// Mitsubishi GX Works2 project: FLASH_EX   PLC: Q03UDV

PROGRAM MAIN
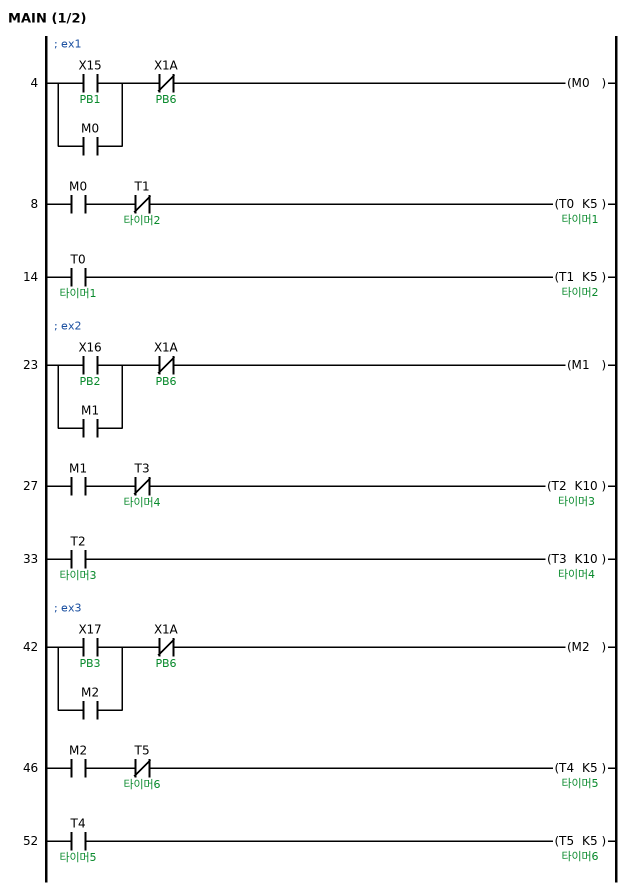
; ex1
4     LD      X15  ; PB1
      OR      M0
      ANI     X1A  ; PB6
      OUT     M0
8     LD      M0
      ANI     T1  ; 타이머2
      OUT     T0 K5  ; 타이머1
14    LD      T0  ; 타이머1
      OUT     T1 K5  ; 타이머2
; ex2
23    LD      X16  ; PB2
      OR      M1
      ANI     X1A  ; PB6
      OUT     M1
27    LD      M1
      ANI     T3  ; 타이머4
      OUT     T2 K10  ; 타이머3
33    LD      T2  ; 타이머3
      OUT     T3 K10  ; 타이머4
; ex3
42    LD      X17  ; PB3
      OR      M2
      ANI     X1A  ; PB6
      OUT     M2
46    LD      M2
      ANI     T5  ; 타이머6
      OUT     T4 K5  ; 타이머5
52    LD      T4  ; 타이머5
      OUT     T5 K5  ; 타이머6
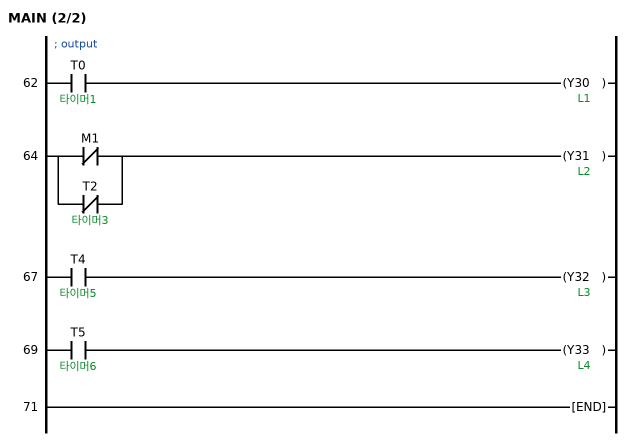
; output
62    LD      T0  ; 타이머1
      OUT     Y30  ; L1
64    LDI     M1
      ORI     T2  ; 타이머3
      OUT     Y31  ; L2
67    LD      T4  ; 타이머5
      OUT     Y32  ; L3
69    LD      T5  ; 타이머6
      OUT     Y33  ; L4
71    END
END_PROGRAM

// device comments not shown above
X19  ; PB6
